GLOBALCONSTANTS Modules_with_medium_IO_density (* Global constants *)
  (* Standard: 61499-1 *)
  (* Version 1.0, 2024-01-25, franz *)
  VAR_GLOBAL CONSTANT
    MI_00 : USINT := 224;
    MI_01 : USINT := 225;
    MI_02 : USINT := 226;
    MI_03 : USINT := 227;
    MI_04 : USINT := 228;
    MI_05 : USINT := 229;
    MI_06 : USINT := 230;
    MI_07 : USINT := 231;
    MI_08 : USINT := 232;
    MI_09 : USINT := 233;
    MI_10 : USINT := 234;
    MI_11 : USINT := 235;
    MI_12 : USINT := 236;
    MI_13 : USINT := 237;
    MI_14 : USINT := 238;
    MI_15 : USINT := 239;
  END_VAR
END_GLOBALCONSTANTS
